DATA_BLOCK "ST10_Flow7_CGlueing_iDB"
VAR
  sCtrlMode : "SysFlowCtrlGraph";
  sUpdMES_Data : Bool;
  "工件放行中" : Bool;
  "前站站号" : UInt;
  "本站站号" : UInt;
  "弹窗Temp" : Array[1..10] of Int;
  AlarmID : Int;
  TON : Array[0..10] of TON_TIME;
  TOF : Array[0..10] of TOF_TIME;
  sUP : Array[0..10] of Bool;
  "更新RFID完成" : Bool;
  RT_DATA : G7_RTDataPlus_V6;
  Trans1 : G7_TransitionPlus_V6;
  Trans2 : G7_TransitionPlus_V6;
  Trans3 : G7_TransitionPlus_V6;
  Trans325 : G7_TransitionPlus_V6;
  Trans4 : G7_TransitionPlus_V6;
  Trans10 : G7_TransitionPlus_V6;
  Trans102 : G7_TransitionPlus_V6;
  Offline : G7_TransitionPlus_V6;
  Offline_1 : G7_TransitionPlus_V6;
  Trans23 : G7_TransitionPlus_V6;
  Trans24 : G7_TransitionPlus_V6;
  Trans25 : G7_TransitionPlus_V6;
  Trans26 : G7_TransitionPlus_V6;
  Trans27 : G7_TransitionPlus_V6;
  NG : G7_TransitionPlus_V6;
  Trans29 : G7_TransitionPlus_V6;
  Trans30 : G7_TransitionPlus_V6;
  Trans36 : G7_TransitionPlus_V6;
  Trans33 : G7_TransitionPlus_V6;
  Trans34 : G7_TransitionPlus_V6;
  Trans37 : G7_TransitionPlus_V6;
  Trans38 : G7_TransitionPlus_V6;
  Trans39 : G7_TransitionPlus_V6;
  Trans40 : G7_TransitionPlus_V6;
  Trans41 : G7_TransitionPlus_V6;
  Trans43 : G7_TransitionPlus_V6;
  Trans44 : G7_TransitionPlus_V6;
  Trans45 : G7_TransitionPlus_V6;
  Trans46 : G7_TransitionPlus_V6;
  Trans47 : G7_TransitionPlus_V6;
  Trans48 : G7_TransitionPlus_V6;
  Trans49 : G7_TransitionPlus_V6;
  Trans50 : G7_TransitionPlus_V6;
  Trans51 : G7_TransitionPlus_V6;
  Trans53 : G7_TransitionPlus_V6;
  Trans54 : G7_TransitionPlus_V6;
  Trans55 : G7_TransitionPlus_V6;
  Trans56 : G7_TransitionPlus_V6;
  Trans57 : G7_TransitionPlus_V6;
  Trans58 : G7_TransitionPlus_V6;
  Trans59 : G7_TransitionPlus_V6;
  Trans60 : G7_TransitionPlus_V6;
  Trans61 : G7_TransitionPlus_V6;
  Trans62 : G7_TransitionPlus_V6;
  Trans63 : G7_TransitionPlus_V6;
  Trans64 : G7_TransitionPlus_V6;
  Trans65 : G7_TransitionPlus_V6;
  Trans66 : G7_TransitionPlus_V6;
  Trans67 : G7_TransitionPlus_V6;
  Trans68 : G7_TransitionPlus_V6;
  Trans69 : G7_TransitionPlus_V6;
  Trans70 : G7_TransitionPlus_V6;
  Trans71 : G7_TransitionPlus_V6;
  Trans72 : G7_TransitionPlus_V6;
  Trans73 : G7_TransitionPlus_V6;
  Trans74 : G7_TransitionPlus_V6;
  Trans75 : G7_TransitionPlus_V6;
  Trans76 : G7_TransitionPlus_V6;
  Trans77 : G7_TransitionPlus_V6;
  Trans78 : G7_TransitionPlus_V6;
  Trans79 : G7_TransitionPlus_V6;
  Trans80 : G7_TransitionPlus_V6;
  Trans83 : G7_TransitionPlus_V6;
  Trans84 : G7_TransitionPlus_V6;
  Trans85 : G7_TransitionPlus_V6;
  Trans86 : G7_TransitionPlus_V6;
  Trans87 : G7_TransitionPlus_V6;
  Trans88 : G7_TransitionPlus_V6;
  Trans89 : G7_TransitionPlus_V6;
  Trans90 : G7_TransitionPlus_V6;
  Trans107 : G7_TransitionPlus_V6;
  Trans31 : G7_TransitionPlus_V6;
  Trans32 : G7_TransitionPlus_V6;
  Trans100 : G7_TransitionPlus_V6;
  Trans105 : G7_TransitionPlus_V6;
  Trans106 : G7_TransitionPlus_V6;
  Trans95 : G7_TransitionPlus_V6;
  Trans97 : G7_TransitionPlus_V6;
  Trans98 : G7_TransitionPlus_V6;
  Trans99 : G7_TransitionPlus_V6;
  Trans103 : G7_TransitionPlus_V6;
  Trans104 : G7_TransitionPlus_V6;
  Trans42 : G7_TransitionPlus_V6;
  Trans108 : G7_TransitionPlus_V6;
  Trans200 : G7_TransitionPlus_V6;
  Trans101 : G7_TransitionPlus_V6;
  Trans109 : G7_TransitionPlus_V6;
  Trans110 : G7_TransitionPlus_V6;
  Trans111 : G7_TransitionPlus_V6;
  Trans112 : G7_TransitionPlus_V6;
  Trans113 : G7_TransitionPlus_V6;
  Trans114 : G7_TransitionPlus_V6;
  Trans122 : G7_TransitionPlus_V6;
  Trans116 : G7_TransitionPlus_V6;
  Trans117 : G7_TransitionPlus_V6;
  Trans118 : G7_TransitionPlus_V6;
  Trans119 : G7_TransitionPlus_V6;
  Trans120 : G7_TransitionPlus_V6;
  Trans115 : G7_TransitionPlus_V6;
  Trans121 : G7_TransitionPlus_V6;
  Trans123 : G7_TransitionPlus_V6;
  Trans126 : G7_TransitionPlus_V6;
  Trans127 : G7_TransitionPlus_V6;
  Trans128 : G7_TransitionPlus_V6;
  Trans767 : G7_TransitionPlus_V6;
  Trans768 : G7_TransitionPlus_V6;
  Trans769 : G7_TransitionPlus_V6;
  Trans770 : G7_TransitionPlus_V6;
  Trans124 : G7_TransitionPlus_V6;
  Trans125 : G7_TransitionPlus_V6;
  Trans129 : G7_TransitionPlus_V6;
  Trans130 : G7_TransitionPlus_V6;
  Trans131 : G7_TransitionPlus_V6;
  Trans132 : G7_TransitionPlus_V6;
  Trans133 : G7_TransitionPlus_V6;
  Trans134 : G7_TransitionPlus_V6;
  Trans135 : G7_TransitionPlus_V6;
  Trans136 : G7_TransitionPlus_V6;
  Trans137 : G7_TransitionPlus_V6;
  Trans138 : G7_TransitionPlus_V6;
  Trans139 : G7_TransitionPlus_V6;
  Trans140 : G7_TransitionPlus_V6;
  Trans141 : G7_TransitionPlus_V6;
  Trans142 : G7_TransitionPlus_V6;
  Trans143 : G7_TransitionPlus_V6;
  Trans144 : G7_TransitionPlus_V6;
  Trans145 : G7_TransitionPlus_V6;
  Trans146 : G7_TransitionPlus_V6;
  Trans147 : G7_TransitionPlus_V6;
  Trans148 : G7_TransitionPlus_V6;
  Trans149 : G7_TransitionPlus_V6;
  Trans150 : G7_TransitionPlus_V6;
  Trans151 : G7_TransitionPlus_V6;
  Trans250 : G7_TransitionPlus_V6;
  Trans161 : G7_TransitionPlus_V6;
  Trans154 : G7_TransitionPlus_V6;
  Trans155 : G7_TransitionPlus_V6;
  Trans156 : G7_TransitionPlus_V6;
  Trans157 : G7_TransitionPlus_V6;
  Trans158 : G7_TransitionPlus_V6;
  Trans159 : G7_TransitionPlus_V6;
  Trans160 : G7_TransitionPlus_V6;
  Trans162 : G7_TransitionPlus_V6;
  Trans163 : G7_TransitionPlus_V6;
  Trans164 : G7_TransitionPlus_V6;
  Trans165 : G7_TransitionPlus_V6;
  Trans166 : G7_TransitionPlus_V6;
  Trans167 : G7_TransitionPlus_V6;
  Trans168 : G7_TransitionPlus_V6;
  Trans169 : G7_TransitionPlus_V6;
  bypassFALSE : G7_TransitionPlus_V6;
  Trans170 : G7_TransitionPlus_V6;
  bypassTRUE : G7_TransitionPlus_V6;
  Trans171 : G7_TransitionPlus_V6;
  Trans35 : G7_TransitionPlus_V6;
  Trans202 : G7_TransitionPlus_V6;
  Trans203 : G7_TransitionPlus_V6;
  Trans205 : G7_TransitionPlus_V6;
  Trans206 : G7_TransitionPlus_V6;
  Trans204 : G7_TransitionPlus_V6;
  Trans207 : G7_TransitionPlus_V6;
  Trans208 : G7_TransitionPlus_V6;
  Trans201 : G7_TransitionPlus_V6;
  Trans81 : G7_TransitionPlus_V6;
  Trans93 : G7_TransitionPlus_V6;
  Trans287 : G7_TransitionPlus_V6;
  Trans82 : G7_TransitionPlus_V6;
  Trans94 : G7_TransitionPlus_V6;
  Trans290 : G7_TransitionPlus_V6;
  Trans286 : G7_TransitionPlus_V6;
  Trans291 : G7_TransitionPlus_V6;
  Online : G7_TransitionPlus_V6;
  Trans259 : G7_TransitionPlus_V6;
  Trans14 : G7_TransitionPlus_V6;
  Online_1 : G7_TransitionPlus_V6;
  Trans264 : G7_TransitionPlus_V6;
  Trans306 : G7_TransitionPlus_V6;
  Trans307 : G7_TransitionPlus_V6;
  Trans15 : G7_TransitionPlus_V6;
  Trans315 : G7_TransitionPlus_V6;
  Trans260 : G7_TransitionPlus_V6;
  Trans610 : G7_TransitionPlus_V6;
  Trans17 : G7_TransitionPlus_V6;
  Trans266 : G7_TransitionPlus_V6;
  Trans301 : G7_TransitionPlus_V6;
  Trans322 : G7_TransitionPlus_V6;
  Trans316 : G7_TransitionPlus_V6;
  Trans317 : G7_TransitionPlus_V6;
  Trans320 : G7_TransitionPlus_V6;
  Trans312 : G7_TransitionPlus_V6;
  Trans313 : G7_TransitionPlus_V6;
  Trans319 : G7_TransitionPlus_V6;
  Trans321 : G7_TransitionPlus_V6;
  Trans326 : G7_TransitionPlus_V6;
  Trans327 : G7_TransitionPlus_V6;
  Trans91 : G7_TransitionPlus_V6;
  Trans311 : G7_TransitionPlus_V6;
  Trans92 : G7_TransitionPlus_V6;
  Trans401 : G7_TransitionPlus_V6;
  Trans613 : G7_TransitionPlus_V6;
  Trans96 : G7_TransitionPlus_V6;
  Trans153 : G7_TransitionPlus_V6;
  Trans152 : G7_TransitionPlus_V6;
  F7_Initial : G7_StepPlus_V6;
  S2 : G7_StepPlus_V6;
  S3 : G7_StepPlus_V6;
  S4 : G7_StepPlus_V6;
  S5_MESInitial : G7_StepPlus_V6;
  "ServoReady?" : G7_StepPlus_V6;
  WaitRobotInitialFinish : G7_StepPlus_V6;
  S10_InitialFinish : G7_StepPlus_V6;
  Axis_YToHomePos : G7_StepPlus_V6;
  "Servo returns toHome Pos" : G7_StepPlus_V6;
  CheckPartStatus : G7_StepPlus_V6;
  StatusAlarm : G7_StepPlus_V6;
  Axis_YToGlueePos_1 : G7_StepPlus_V6;
  RequestRobot1PutShaft : G7_StepPlus_V6;
  WaitRobot1FinishTask : G7_StepPlus_V6;
  Axis_XToGluePos_1 : G7_StepPlus_V6;
  CheckGlueSysOK : G7_StepPlus_V6;
  "Servo returns toGluePos_1" : G7_StepPlus_V6;
  Axis_XToGlueSafPos : G7_StepPlus_V6;
  Glue_1 : G7_StepPlus_V6;
  Axis_ZToGlueePos_2 : G7_StepPlus_V6;
  Axis_XToGluePos_2 : G7_StepPlus_V6;
  CheckGlueSysOK_1 : G7_StepPlus_V6;
  "Servo returns toGluePos_2" : G7_StepPlus_V6;
  Axis_XToGlueSafPos_2 : G7_StepPlus_V6;
  Glue_2 : G7_StepPlus_V6;
  Axis_YToGlueePos_5 : G7_StepPlus_V6;
  TimeDelay_1 : G7_StepPlus_V6;
  TimeDelay_2 : G7_StepPlus_V6;
  Axis_ZToGlueePos_3 : G7_StepPlus_V6;
  Axis_XToGluePos_3 : G7_StepPlus_V6;
  CheckGlueSysOK_2 : G7_StepPlus_V6;
  "Servo returns toGluePos_3" : G7_StepPlus_V6;
  Axis_XToGlueSafPos_3 : G7_StepPlus_V6;
  Glue_3 : G7_StepPlus_V6;
  TimeDelay_3 : G7_StepPlus_V6;
  Axis_YToGlueePos_6 : G7_StepPlus_V6;
  Axis_ZToGlueePos_4 : G7_StepPlus_V6;
  Axis_XToGluePos_4 : G7_StepPlus_V6;
  CheckGlueSysOK_3 : G7_StepPlus_V6;
  "Servo returns toGluePos_4" : G7_StepPlus_V6;
  Axis_XToGlueSafPos_4 : G7_StepPlus_V6;
  Glue_4 : G7_StepPlus_V6;
  TimeDelay_4 : G7_StepPlus_V6;
  IV3Check : G7_StepPlus_V6;
  JudgeCheckStatus : G7_StepPlus_V6;
  OKStatus : G7_StepPlus_V6;
  NGStatus : G7_StepPlus_V6;
  PutMagnet : G7_StepPlus_V6;
  Magnet_Glue : G7_StepPlus_V6;
  Magnet_GlueCheck : G7_StepPlus_V6;
  "Shaft GlueCheck" : G7_StepPlus_V6;
  ShaftGlueFinishStatus : G7_StepPlus_V6;
  IV3Check_1 : G7_StepPlus_V6;
  Axis_ZToGlueePos_5 : G7_StepPlus_V6;
  Axis_XToGluePos_5 : G7_StepPlus_V6;
  CheckGlueSysOK_4 : G7_StepPlus_V6;
  "Servo returns toGluePos_5" : G7_StepPlus_V6;
  JudgeCheckStatus_1 : G7_StepPlus_V6;
  Axis_YToGluePos_5 : G7_StepPlus_V6;
  TimeDelay_5 : G7_StepPlus_V6;
  Axis_ZToIVCheckPos : G7_StepPlus_V6;
  Axis_XYIVCheckPos : G7_StepPlus_V6;
  Axis_ZToHomePos_1 : G7_StepPlus_V6;
  Axis_XToHomePos : G7_StepPlus_V6;
  Axis_ZToHomePos_2 : G7_StepPlus_V6;
  GlueFinishStatus : G7_StepPlus_V6;
  OKStatus_1 : G7_StepPlus_V6;
  NGStatus_1 : G7_StepPlus_V6;
  Axis_XYToHomePos_1 : G7_StepPlus_V6;
  Step87 : G7_StepPlus_V6;
  Axis_YToGlueePos_7 : G7_StepPlus_V6;
  Axis_ZToGlueePos_1 : G7_StepPlus_V6;
  JudgeYPosition : G7_StepPlus_V6;
  Axis_YToGluePos_6 : G7_StepPlus_V6;
  Axis_XToGluePos_6 : G7_StepPlus_V6;
  Axis_ZToGlueePos_6 : G7_StepPlus_V6;
  ServoHomePos : G7_StepPlus_V6;
  IAIMoveFinish : G7_StepPlus_V6;
  GluePos_1 : G7_StepPlus_V6;
  ServoHomePos_1 : G7_StepPlus_V6;
  GluePos_2 : G7_StepPlus_V6;
  "CheckServo returns toHome Pos_5" : G7_StepPlus_V6;
  ProcessStart : G7_StepPlus_V6;
  "WaitTableCode OK" : G7_StepPlus_V6;
  Step102 : G7_StepPlus_V6;
  WaitIAIStop : G7_StepPlus_V6;
  Step104 : G7_StepPlus_V6;
  IAIMoveFinish_1 : G7_StepPlus_V6;
  WaitIAIStop_1 : G7_StepPlus_V6;
  Step107 : G7_StepPlus_V6;
  IAIMoveFinish_2 : G7_StepPlus_V6;
  WaitIAIStop_2 : G7_StepPlus_V6;
  Step110 : G7_StepPlus_V6;
  IAIMoveFinish_3 : G7_StepPlus_V6;
  WaitIAIStop_3 : G7_StepPlus_V6;
  ServoHomePos_2 : G7_StepPlus_V6;
  GluePos_3 : G7_StepPlus_V6;
  ServoHomePos_3 : G7_StepPlus_V6;
  GluePos_4 : G7_StepPlus_V6;
  ServoHomePos_4 : G7_StepPlus_V6;
  CameraCheck1 : G7_StepPlus_V6;
  "C-LocationCylinderToHP" : G7_StepPlus_V6;
  "C-LocationCylinderToWP_1" : G7_StepPlus_V6;
  "C-LocationCylinderToWP_2" : G7_StepPlus_V6;
  "C-LocationCylinderToHP2" : G7_StepPlus_V6;
  ServoJoging : G7_StepPlus_V6;
  StopServoJoging : G7_StepPlus_V6;
  "Servo returns toGluePos_6" : G7_StepPlus_V6;
  CameraCheck2 : G7_StepPlus_V6;
  IV3Check_2 : G7_StepPlus_V6;
  JudgeCheckStatus_2 : G7_StepPlus_V6;
  OKStatus_2 : G7_StepPlus_V6;
  NGStatus_2 : G7_StepPlus_V6;
  CameraCheck3 : G7_StepPlus_V6;
  "Servo returns toGluePos_7" : G7_StepPlus_V6;
  IV3Check_3 : G7_StepPlus_V6;
  JudgeCheckStatus_3 : G7_StepPlus_V6;
  OKStatus_3 : G7_StepPlus_V6;
  NGStatus_3 : G7_StepPlus_V6;
  CameraCheck4 : G7_StepPlus_V6;
  "Servo returns toGluePos_8" : G7_StepPlus_V6;
  IV3Check_4 : G7_StepPlus_V6;
  JudgeCheckStatus_4 : G7_StepPlus_V6;
  OKStatus_4 : G7_StepPlus_V6;
  NGStatus_4 : G7_StepPlus_V6;
  ServoHomePos_5 : G7_StepPlus_V6;
  ServoHomePos_6 : G7_StepPlus_V6;
  Step145 : G7_StepPlus_V6;
  Step146 : G7_StepPlus_V6;
  CheckAxisXPos : G7_StepPlus_V6;
  Axis_ZToGlueePos_7 : G7_StepPlus_V6;
  "Process Finish" : G7_StepPlus_V6;
  "MES Check" : G7_StepPlus_V6;
  MESResult : G7_StepPlus_V6;
  OKPart : G7_StepPlus_V6;
  "IAIMoveFinish_ 1" : G7_StepPlus_V6;
  IAIMoveFinish_5 : G7_StepPlus_V6;
  IAIMoveFinish_4 : G7_StepPlus_V6;
  Axis_XYToHomePos_2 : G7_StepPlus_V6;
  Axis_XYIVCheckPos_1 : G7_StepPlus_V6;
  Step158 : G7_StepPlus_V6;
  Step159 : G7_StepPlus_V6;
  Step160 : G7_StepPlus_V6;
  Step161 : G7_StepPlus_V6;
  bypassGlue4 : G7_StepPlus_V6;
  Glue2s : G7_StepPlus_V6;
  ShaftGluingProcess : G7_StepPlus_V6;
  CheckIV3Ready : G7_StepPlus_V6;
  Step203 : G7_StepPlus_V6;
  CheckIV3Ready_1 : G7_StepPlus_V6;
  Step204 : G7_StepPlus_V6;
  CheckIV3Ready_2 : G7_StepPlus_V6;
  CheckIV3Ready_3 : G7_StepPlus_V6;
  CheckIV3Ready_4 : G7_StepPlus_V6;
  ShaftGlueCameraCheck : G7_StepPlus_V6;
  RequestRobotPutMagnet_1 : G7_StepPlus_V6;
  RequestRobotGluePick : G7_StepPlus_V6;
  "Shaft Glue" : G7_StepPlus_V6;
  WaitRobotFinishTask_1 : G7_StepPlus_V6;
  WaitRobotFinishTask_2 : G7_StepPlus_V6;
  "Process  Finish" : G7_StepPlus_V6;
  ShaftGlueProcessFinish : G7_StepPlus_V6;
  RobotPutMagnet : G7_StepPlus_V6;
  ResetMesCheckRequest : G7_StepPlus_V6;
  ResetMesCheckRequest_1 : G7_StepPlus_V6;
  "Prepare MES CheckData" : G7_StepPlus_V6;
  "MES Check OK" : G7_StepPlus_V6;
  "Prepare MES CheckData_1" : G7_StepPlus_V6;
  MESCheckRequest : G7_StepPlus_V6;
  ok : G7_StepPlus_V6;
  MESSaveRequest_1 : G7_StepPlus_V6;
  Bypass : G7_StepPlus_V6;
  "Check OK" : G7_StepPlus_V6;
  "Check NG" : G7_StepPlus_V6;
  MESOverTime_1 : G7_StepPlus_V6;
  MaganetGlue : G7_StepPlus_V6;
  Step314 : G7_StepPlus_V6;
  MESOverTime : G7_StepPlus_V6;
  Bypass_1 : G7_StepPlus_V6;
  ResultNG : G7_StepPlus_V6;
  Step315 : G7_StepPlus_V6;
  ok_1 : G7_StepPlus_V6;
  MagnetGlueFinish : G7_StepPlus_V6;
  "MES  Check Result" : G7_StepPlus_V6;
  "MES Check OK_1" : G7_StepPlus_V6;
  RobotGluePick : G7_StepPlus_V6;
  PartNG : G7_StepPlus_V6;
  "IV3 Check" : G7_StepPlus_V6;
END_VAR
BEGIN
END_DATA_BLOCK
